Omron Sysmac Studio project modbus_tcp_ok_plc_s7_1200_ss1 (Sysmac Studio 1.45.1.64010, StandardProject)

# Controller new_Controller_0: NX1P2-9024DT version 1.40
Units and slaves: Node86 : NX-ECC201 (E001); Unit 1 : NX-OD5121 (N1); Unit 2 : NX-OD4256 (N2); Unit 3 : NX-ID5342 (N3); Unit 4 : NX-ID5442 (N4); Node1 : GX-ID1611+OD16 (E002)
Task PrimaryTask (priority 4, period or condition 2000): Program0
Library OEN_Communication_V1_0_22 1.0.22 (contents left out)

VAR_GLOBAL
    NX1P2_OUT_0 : BOOL;  (* output_nx1p2; at BuiltInIO://cpu/#0/Output_Bit_00 *)
    NX1P2_OUT_1 : BOOL;  (* output_nx1p2; at BuiltInIO://cpu/#0/Output_Bit_01 *)
    NX1P2_OUT_2 : BOOL;  (* output_nx1p2; at BuiltInIO://cpu/#0/Output_Bit_02 *)
    NX1P2_OUT_3 : BOOL;  (* output_nx1p2; at BuiltInIO://cpu/#0/Output_Bit_03 *)
    NX1P2_OUT_4 : BOOL;  (* output_nx1p2; at BuiltInIO://cpu/#0/Output_Bit_04 *)
    NX1P2_OUT_5 : BOOL;  (* output_nx1p2; at BuiltInIO://cpu/#0/Output_Bit_05 *)
    NX1P2_OUT_6 : BOOL;  (* output_nx1p2; at BuiltInIO://cpu/#0/Output_Bit_06 *)
    NX1P2_OUT_7 : BOOL;  (* output_nx1p2; at BuiltInIO://cpu/#0/Output_Bit_07 *)
    NX1P2_OUT_8 : BOOL;  (* output_nx1p2; at BuiltInIO://cpu/#0/Output_Bit_08 *)
    NX1P2_OUT_9 : BOOL;  (* output_nx1p2; at BuiltInIO://cpu/#0/Output_Bit_09 *)
    NX1P2_IN_0 : BOOL;  (* INPUT_NX1P2_9024DT; at BuiltInIO://cpu/#0/Input_Bit_00 *)
    NX1P2_IN_1 : BOOL;  (* INPUT_NX1P2_9024DT; at BuiltInIO://cpu/#0/Input_Bit_01 *)
    NX1P2_IN_2 : BOOL;  (* INPUT_NX1P2_9024DT; at BuiltInIO://cpu/#0/Input_Bit_02 *)
    NX1P2_IN_3 : BOOL;  (* INPUT_NX1P2_9024DT; at BuiltInIO://cpu/#0/Input_Bit_03 *)
    NX1P2_IN_4 : BOOL;  (* INPUT_NX1P2_9024DT; at BuiltInIO://cpu/#0/Input_Bit_04 *)
    NX1P2_IN_5 : BOOL;  (* INPUT_NX1P2_9024DT; at BuiltInIO://cpu/#0/Input_Bit_05 *)
    NX1P2_IN_6 : BOOL;  (* INPUT_NX1P2_9024DT; at BuiltInIO://cpu/#0/Input_Bit_06 *)
    NX1P2_IN_7 : BOOL;  (* INPUT_NX1P2_9024DT; at BuiltInIO://cpu/#0/Input_Bit_07 *)
    NX1P2_IN_8 : BOOL;  (* INPUT_NX1P2_9024DT; at BuiltInIO://cpu/#0/Input_Bit_08 *)
    NX1P2_IN_9 : BOOL;  (* INPUT_NX1P2_9024DT; at BuiltInIO://cpu/#0/Input_Bit_09 *)
    NX1P2_IN_10 : BOOL;  (* INPUT_NX1P2_9024DT; at BuiltInIO://cpu/#0/Input_Bit_10 *)
    NX1P2_IN_11 : BOOL;  (* INPUT_NX1P2_9024DT; at BuiltInIO://cpu/#0/Input_Bit_11 *)
    NX1P2_IN_12 : BOOL;  (* INPUT_NX1P2_9024DT; at BuiltInIO://cpu/#0/Input_Bit_12 *)
    NX1P2_IN_13 : BOOL;  (* INPUT_NX1P2_9024DT; at BuiltInIO://cpu/#0/Input_Bit_13 *)
END_VAR

PROGRAM Program0
VAR
    TCP_SERVER_CONNECT : BOOL;
    FB_TCP_SERVER : OEN\Modbus\ModbusTCP_Server;
    DATA_ACCESS_LIST : ARRAY[0..0] OF OEN\Modbus\sModbusAccess := [(RegisterType := Coil, AccessType := R, AddressArea := (StartAddress := 0, Count := 0))];
    MODBUS_COIL : ARRAY[0..16] OF BOOL;
    DISCRETE_INPUT : ARRAY[0..10] OF BOOL;
    MODBUS_DISCRETE_INPUT : ARRAY[0..10] OF BOOL;
    INPUT_RES : ARRAY[0..10] OF WORD;
    HOLDING_REGISTER : ARRAY[0..20] OF WORD;
    TRANSFER_RES : ARRAY[0..11] OF WORD;
    T0_TCP : TON;
    T1_TCP : TON;
    TCP_SERVER_DISCONNECT : BOOL;
    READ_DATA_TCP : ARRAY[0..9] OF WORD;
    WRITE_DATA_TCP : ARRAY[0..9] OF WORD;
    INT_DATA_WRITE : ARRAY[0..9] OF INT;
    INT_DATA_READ : ARRAY[0..9] OF INT;
    T0 : TON;
    T1 : TON;
    T3 : TON;
    T2 : TON;
    T4 : TON;
    T5 : TON;
    T6 : TON;
    T7 : TON;
    i : int;
    i1 : int;
END_VAR
VAR_EXTERNAL
    NX1P2_OUT_0 : BOOL;
    NX1P2_OUT_1 : BOOL;
    NX1P2_IN_0 : BOOL;
    NX1P2_IN_1 : BOOL;
    NX1P2_IN_2 : BOOL;
    NX1P2_OUT_2 : BOOL;
    NX1P2_OUT_3 : BOOL;
    NX1P2_OUT_4 : BOOL;
    NX1P2_IN_3 : BOOL;
    NX1P2_IN_4 : BOOL;
END_VAR
VAR
    _e1 : R_TRIG;
    _e2 : R_TRIG;
    _e3 : R_TRIG;
    _e4 : R_TRIG;
    _e5 : R_TRIG;
END_VAR

(* Section Section0: ladder, written here as Structured Text *)

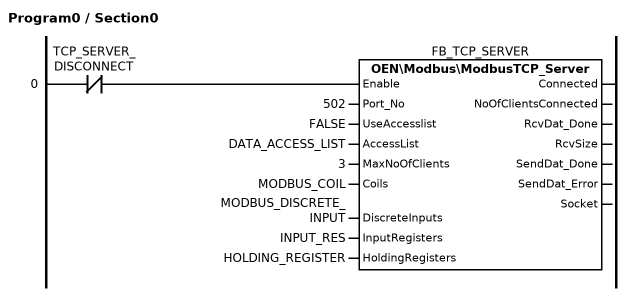
(* Rung 0 *)
FB_TCP_SERVER(Enable := NOT TCP_SERVER_DISCONNECT, Port_No := 502, UseAccesslist := FALSE, AccessList := DATA_ACCESS_LIST, MaxNoOfClients := 3, Coils := MODBUS_COIL, DiscreteInputs := MODBUS_DISCRETE_INPUT, InputRegisters := INPUT_RES, HoldingRegisters := HOLDING_REGISTER);

(* Section write_data_tcp: ladder, written here as Structured Text *)

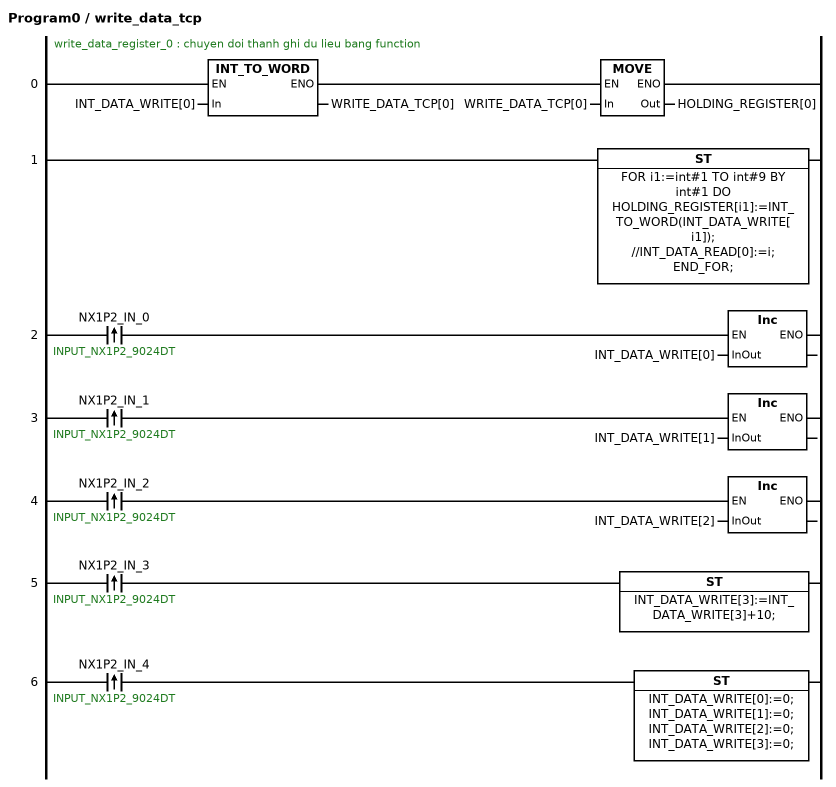
(* Rung 0: write_data_register_0 : chuyen doi thanh ghi du lieu bang function *)
WRITE_DATA_TCP[0] := INT_TO_WORD(In := INT_DATA_WRITE[0]);
HOLDING_REGISTER[0] := WRITE_DATA_TCP[0];
(* Rung 1 *)
FOR i1:=int#1 TO int#9 BY int#1 DO
	 HOLDING_REGISTER[i1]:=INT_TO_WORD(INT_DATA_WRITE[i1]);
	 //INT_DATA_READ[0]:=i;
 END_FOR;
(* Rung 2 *)
_e1(CLK := NX1P2_IN_0);
IF _e1.Q THEN Inc(InOut := INT_DATA_WRITE[0]); END_IF;
(* Rung 3 *)
_e2(CLK := NX1P2_IN_1);
IF _e2.Q THEN Inc(InOut := INT_DATA_WRITE[1]); END_IF;
(* Rung 4 *)
_e3(CLK := NX1P2_IN_2);
IF _e3.Q THEN Inc(InOut := INT_DATA_WRITE[2]); END_IF;
(* Rung 5 *)
_e4(CLK := NX1P2_IN_3);
IF _e4.Q THEN
    INT_DATA_WRITE[3]:=INT_DATA_WRITE[3]+10;
END_IF;
(* Rung 6 *)
_e5(CLK := NX1P2_IN_4);
IF _e5.Q THEN
    INT_DATA_WRITE[0]:=0;
    INT_DATA_WRITE[1]:=0;
    INT_DATA_WRITE[2]:=0;
    INT_DATA_WRITE[3]:=0;
END_IF;

(* Section read_data: ladder, written here as Structured Text *)

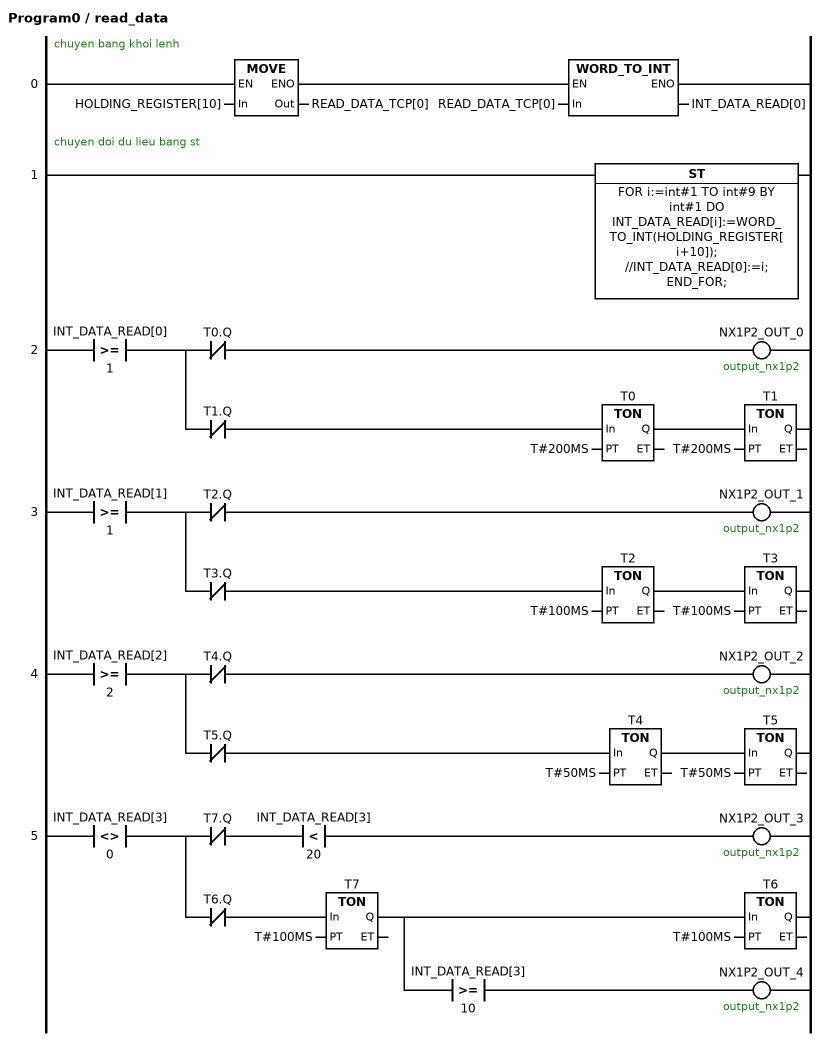
(* Rung 0: chuyen bang khoi lenh *)
READ_DATA_TCP[0] := HOLDING_REGISTER[10];
INT_DATA_READ[0] := WORD_TO_INT(In := READ_DATA_TCP[0]);
(* Rung 1: chuyen doi du lieu bang st *)
FOR i:=int#1 TO int#9 BY int#1 DO
	 INT_DATA_READ[i]:=WORD_TO_INT(HOLDING_REGISTER[i+10]);
	 //INT_DATA_READ[0]:=i;
 END_FOR;
(* Rung 2 *)
NX1P2_OUT_0 := (INT_DATA_READ[0] >= 1) AND NOT T0.Q;
T0(In := (INT_DATA_READ[0] >= 1) AND NOT T1.Q, PT := T#200MS);
T1(In := T0.Q, PT := T#200MS);
(* Rung 3 *)
NX1P2_OUT_1 := (INT_DATA_READ[1] >= 1) AND NOT T2.Q;
T2(In := (INT_DATA_READ[1] >= 1) AND NOT T3.Q, PT := T#100MS);
T3(In := T2.Q, PT := T#100MS);
(* Rung 4 *)
NX1P2_OUT_2 := (INT_DATA_READ[2] >= 2) AND NOT T4.Q;
T4(In := (INT_DATA_READ[2] >= 2) AND NOT T5.Q, PT := T#50MS);
T5(In := T4.Q, PT := T#50MS);
(* Rung 5 *)
NX1P2_OUT_3 := (INT_DATA_READ[3] <> 0) AND NOT T7.Q AND (INT_DATA_READ[3] < 20);
T7(In := (INT_DATA_READ[3] <> 0) AND NOT T6.Q, PT := T#100MS);
T6(In := T7.Q, PT := T#100MS);
NX1P2_OUT_4 := T7.Q AND (INT_DATA_READ[3] >= 10);
END_PROGRAM